(* IEC 61131-3 sources: Chopper/, 3 files *)

(* ---- Types.typ ---- *)
TYPE
	Chop_Status_Enum :
		(
		CHOP_ERR_INVALID_INPUT := 50000,
		CHOP_ERR_SOURCE_LENGTH,
		CHOP_ERR_TEMPLATE_FULL,
		CHOP_ERR_NO_END_OF_VAR, (*Check source vars are surrounded by '{{}}'*)
		CHOP_ERR_NOT_COMPILED,
		CHOP_ERR_DEST_LENGTH, (*50005*)
		CHOP_ERR_INTERNAL,
		CHOP_ERR_INVALID_FORMATTER := 51000 (*51XXX Invalid variable format XXX represents the index of the variable *)
		);
	Chop_Template_typ : 	STRUCT
		snippet : ARRAY[0..CHOP_TEMPLATE_MAI_VARIABLES]OF Chop_Template_Variable_typ;
		iSnippet : UINT;
		source : STRING[CHOP_TEMPLATE_STRLEN_SOURCE];
		compiled : BOOL;
	END_STRUCT;
	Chop_Template_Variable_typ : 	STRUCT
		pv : varVariable_typ;
		prefixStart : UDINT;
		prefixLen : UDINT;
		flags : STRING[CHOP_NUM_FLAG_LEN];
		hasVar : BOOL;
	END_STRUCT;
END_TYPE

(* ---- Chopper.fun ---- *)
FUNCTION ChopCompile : DINT
	VAR_INPUT
		pTemplate : UDINT; (*Address of Template*)
		pSource : UDINT; (*Address of Source*)
	END_VAR
END_FUNCTION

FUNCTION ChopRender : DINT
	VAR_INPUT
		pDest : UDINT;
		pTemplate : UDINT;
		maxDestLength : UDINT;
		pRenderLength : UDINT;
	END_VAR
END_FUNCTION

FUNCTION_BLOCK Chopper
	VAR_INPUT
		pDest : UDINT;
		pTemplate : UDINT;
		pSource : UDINT;
		maxDestLength : UDINT;
		recompile : BOOL;
	END_VAR
	VAR_OUTPUT
		renderLength : UDINT;
		status : DINT;
	END_VAR
	VAR
		compileStatus : DINT;
	END_VAR
END_FUNCTION_BLOCK

FUNCTION ChopReplace : DINT
	VAR_INPUT
		pTemplate : UDINT;
		pTag : UDINT;
		address : UDINT;
		type : UDINT;
	END_VAR
END_FUNCTION

FUNCTION ChopReplaceVar : DINT
	VAR_INPUT
		pTemplate : UDINT;
		pTag : UDINT;
		pVarName : UDINT;
	END_VAR
END_FUNCTION
(*--- Utility Fns ---*)

FUNCTION ChopGetErrorMsg : DINT
	VAR_INPUT
		pDest : UDINT;
		maxDestLength : UDINT;
		errorID : DINT;
	END_VAR
END_FUNCTION

FUNCTION ChopGetDefaultFormatter : BOOL
	VAR_INPUT
		dest : STRING[80];
		type : UDINT; (*VAR_TYPE_enum*)
	END_VAR
END_FUNCTION

FUNCTION ChopVerifyFormatter : BOOL
	VAR_INPUT
		pSrc : STRING[80];
		type : UDINT; (*VAR_TYPE_enum*)
	END_VAR
END_FUNCTION

(* ---- Constants.var ---- *)
VAR CONSTANT
	CHOP_NUM_FLAG_LEN : USINT := 30;
	CHOP_TEMPLATE_MAX_VARIABLES : USINT := 100;
	CHOP_TEMPLATE_MAI_VARIABLES : USINT := CHOP_TEMPLATE_MAX_VARIABLES-1;
	CHOP_TEMPLATE_STRLEN_SOURCE : UINT := 5000;
END_VAR
